TYPE ST_MO1008_DI EXTENDS ST_EFU_Data :
STRUCT
	InputStatus			AT%I*	: ST_DIS_Inputs 	;
	InputDiagnostics	AT%I*	: ST_DIS_Diagnosis	;
	ModuleDiagnostics	: ST_EFU_Data		; 
END_STRUCT
END_TYPE

(* stored: Version 1.1.0.1
   DUT ST_MO1008_DI: Id {bd741172-9d4c-4e3e-8f6d-bfbe4ccfa943} *)
